PROGRAM MAIN
VAR
END_VAR


	PRG_House();

END_PROGRAM

(* stored: Version 1.1.0.1, ProductVersion 3.1.4024.13
   POU MAIN: Id {4aa391a1-51d8-43de-b7a4-8fe077caf324}, SpecialFunc None *)
